TYPE ST_FeedbackMru :
STRUCT
	eta: ARRAY[0..5] OF LREAL;
	v: ARRAY[0..5] OF LREAL;
END_STRUCT
END_TYPE

(* stored: Version 1.1.0.1, ProductVersion 3.1.4026.8
   DUT ST_FeedbackMru: Id {69b5770d-2a8c-4ec4-ae8d-3a67e65402de} *)
